ADAPTER IFeeding2 (* Adapter Interface *)
  (* Standard: 61499-1 *)
  (* Version 0.0, 6/7/2026, Schneider Electric *)
  PACKAGE SE.Nereda;
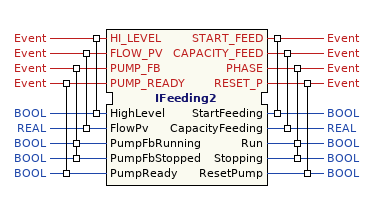
  EVENT_INPUT
    HI_LEVEL WITH HighLevel; (* Request from Socket *)
    FLOW_PV WITH FlowPv; (* Response from Socket *)
    PUMP_FB WITH PumpFbRunning, PumpFbStopped;
    PUMP_READY WITH PumpReady;
  END_EVENT
  EVENT_OUTPUT
    START_FEED WITH StartFeeding; (* Confirmation from Plug *)
    CAPACITY_FEED WITH CapacityFeeding; (* Indication from Plug *)
    PHASE WITH Run, Stopping;
    RESET_P WITH ResetPump;
  END_EVENT
  VAR_INPUT
    HighLevel : BOOL; (* Request Data from Socket *)
    FlowPv : REAL; (* Response Data from Socket *)
    PumpFbRunning : BOOL;
    PumpFbStopped : BOOL;
    PumpReady : BOOL;
  END_VAR
  VAR_OUTPUT
    StartFeeding : BOOL; (* Confirmation Data from Plug *)
    CapacityFeeding : REAL; (* Indication Data from Plug *)
    Run : BOOL;
    Stopping : BOOL;
    ResetPump : BOOL;
  END_VAR
  SERVICE SOCKET/PLUG
    SEQUENCE request_confirm
      SOCKET.HI_LEVEL(HighLevel) -> PLUG.HI_LEVEL(HighLevel);
      PLUG.START_FEED(StartFeeding) -> SOCKET.START_FEED(StartFeeding);
    END_SEQUENCE
    SEQUENCE indication_response
      PLUG.CAPACITY_FEED(CapacityFeeding) -> SOCKET.CAPACITY_FEED(CapacityFeeding);
      SOCKET.FLOW_PV(FlowPv) -> PLUG.FLOW_PV(FlowPv);
    END_SEQUENCE
  END_SERVICE
END_ADAPTER
